FUNCTION_BLOCK ABSTRACT ChuckBase EXTENDS TExecution IMPLEMENTS IDevice
VAR_INPUT
END_VAR
VAR_OUTPUT
END_VAR
VAR
	{attribute 'OPC.UA.DA' := '0'}
	_name : STRING;
	{attribute 'OPC.UA.DA' := '0'}
	_deviceID : STRING;				
	{attribute 'OPC.UA.DA' := '0'}
	_family : DeviceFamily := DeviceFamily.Chuck;		
	{attribute 'OPC.UA.DA' := '0'}
	_logger : Logger;
	{attribute 'OPC.UA.DA' := '0'}
	_message : StringBuilder;
	{attribute 'OPC.UA.DA' := '0'}
	_chuckConfig : DeviceConfiguration;
	
	{attribute 'OPC.UA.DA' := '0'}
	_lifeTimeCount : UINT;
	{attribute 'OPC.UA.DA' := '0'}
	_notifyIsAlive : BOOL;
	{attribute 'OPC.UA.DA' := '0'}
	_pulseIsAliveGenerator : TON;
	{attribute 'OPC.UA.DA' := '0'}
	_pulseGeneratorBase : TON;
	{attribute 'OPC.UA.DA' := '0'}
	_execPulseGeneratorBase : TON;	
	
	{attribute 'OPC.UA.DA' := '0'}
	_itemSchedulerBase : INT;
	{attribute 'OPC.UA.DA' := '0'}
	_itemExecSchedulerBase : INT;	
	
	{attribute 'OPC.UA.DA' := '0'}
	_deliverMessagesBase : INT;
	
	{attribute 'OPC.UA.DA' := '0'}
	_chuckInLoadingPositionCmd : BOOL;
	
	StateMsg : STRING(255);
	IsAliveMsg : STRING(255);
	IsInLoadingPositionMsg : STRING(255);
	
	{attribute 'OPC.UA.DA' := '0'}
	_isInLoadingPosition : BOOL;
	{attribute 'OPC.UA.DA' := '0'}
	_loadingPosition : BOOL;		
	{attribute 'OPC.UA.DA' := '0'}
	IsInLoadingPosition AT %Q* : BOOL;
	
	{attribute 'OPC.UA.DA' := '0'}	
	_waferSize : EWaferSize := EWaferSize.Unknown; 
	
	{attribute 'OPC.UA.DA' := '0'}
	ioMessage : STRING;
END_VAR

// Check if it's still alive	
IF _notifyIsAlive THEN
	IsAliveMsg := TO_STRING(_lifeTimeCount);
	_notifyIsAlive := FALSE;
END_IF

IF HardwareGlobalVariables.ChuckState <> State THEN
	HardwareGlobalVariables.ChuckState := State;
	StateMsg := ANY_TO_STRING(State);		
END_IF

CASE _deliverMessagesBase OF		
	EFeedbackMsgChuckBase.IsInLoadingPositionMsg :	
		IsInLoadingPositionMsg := ioMessage;		
END_CASE

ChuckInLoadingPosition(_chuckInLoadingPositionCmd, _loadingPosition);

IF NOT _chuckInLoadingPositionCmd THEN
	MessageSchedulerBase();	
END_IF

{attribute 'TcRpcEnable' := '1'}
METHOD ChuckInLoadingPosition
VAR_INPUT
	Execute : BOOL;
	LoadingPosition : BOOL;
END_VAR

VAR
	_config: INT;
END_VAR
IF Execute THEN	
	_logger.Information(_message.Reset().Append('ChuckInLoadingPosition: ').Append(TO_STRING(LoadingPosition)).ToString());
	
	IsInLoadingPosition := LoadingPosition;
	_chuckInLoadingPositionCmd := FALSE;
END_IF
END_METHOD

PROPERTY DeviceID : STRING
GET
DeviceID := _deviceID;
END_GET
SET
_deviceID := DeviceID;
END_SET
END_PROPERTY

PROPERTY Family : DeviceFamily
GET
Family := _family;
END_GET
SET
_family := Family;
END_SET
END_PROPERTY

METHOD PROTECTED IsAlive
VAR_INPUT
END_VAR
_notifyIsAlive := TRUE;

IF _lifeTimeCount < 5 THEN
	_lifeTimeCount := _lifeTimeCount + 1;
ELSE
	_lifeTimeCount := 1;
END_IF
END_METHOD

METHOD MessageSchedulerBase
VAR_INPUT
END_VAR
IF _pulseGeneratorBase.Q THEN
	_pulseGeneratorBase(IN := FALSE, PT := T#10MS);
		
	CASE _itemSchedulerBase OF			
		0:  _deliverMessagesBase := EFeedbackMsgChuckBase.IsInLoadingPositionMsg;
			ioMessage := ' ';
			_itemSchedulerBase := 1;
			
		1: _deliverMessagesBase := EFeedbackMsgChuckBase.IsInLoadingPositionMsg;
			ioMessage := TO_STRING(IsInLoadingPosition);
			_itemSchedulerBase := 0;
	END_CASE
ELSE
	_pulseGeneratorBase(IN := TRUE, PT := T#100MS);		
END_IF


IF _pulseIsAliveGenerator.Q THEN
	_pulseIsAliveGenerator(IN := FALSE, PT := T#10MS);
		
	IsAlive();	
ELSE
	_pulseIsAliveGenerator(IN := TRUE, PT := T#1000MS);		
END_IF
END_METHOD

PROPERTY Name : STRING
GET
Name := _name;
END_GET
SET
_name := Name;
END_SET
END_PROPERTY

PROPERTY WaferSize : EWaferSize
GET
WaferSize := _waferSize;
END_GET
SET
_waferSize := WaferSize;
END_SET
END_PROPERTY

END_FUNCTION_BLOCK

(* stored: Version 1.1.0.1, ProductVersion 3.1.4024.12
   POU ChuckBase: Id {8a64419b-624a-4206-9ee2-86d1dbd9bb98}, SpecialFunc None
   Folder Commands: Id {f76c5636-5710-4d49-bb60-31627b9311b9}
   Method ChuckInLoadingPosition: Id {0f9e48b5-78b3-4b8e-b2c2-f5db3200b82a}
   Property DeviceID: Id {f852fc02-d39a-4bf5-8e6d-4848990d040f}
   Get Get: Id {1f3081dc-2999-49d1-81d2-095303c93992}
   Set Set: Id {4f026f99-3695-40ad-b692-bb895065fd84}
   Property Family: Id {588a7060-a055-4d9a-8114-b9d3b8f3e268}
   Get Get: Id {ed432400-b099-44ec-93bd-26caf073b109}
   Set Set: Id {3354990e-5506-4e79-8c76-fd8733e4d4e7}
   Method IsAlive: Id {8a33ad11-1200-4056-997b-43110f8c43e1}
   Method MessageSchedulerBase: Id {b29827ac-3f16-4260-9eab-1729f39c013f}
   Property Name: Id {0ed3b1a0-7cf5-4488-a675-9d95986087e7}
   Get Get: Id {3f4cd8ce-28d9-4f70-ae18-747a667658ba}
   Set Set: Id {227b9f5e-5e5d-4918-87bf-2829008f4401}
   Property WaferSize: Id {d5aabc35-9e6b-4965-a694-8bde647fd5d6}
   Get Get: Id {be0aab99-3136-495c-bbff-6bdcbe97f622}
   Set Set: Id {9febcd9e-54ae-4e74-a623-b792d2347273} *)
